FUNCTION Concat2 : T_MaxString
VAR_INPUT
	sExpression1: T_maxString;
	sExpression2: T_maxString;
END_VAR

Concat2 := CONCAT(sExpression1, sExpression2);

END_FUNCTION

(* stored: Version 1.1.0.1
   POU Concat2: Id {5a9bda90-645e-416f-883f-c90ac3cb0c2d}, SpecialFunc None *)
